FUNCTION_BLOCK ToteData
VAR_INPUT
	
END_VAR
VAR_OUTPUT
END_VAR
VAR_IN_OUT
	
END_VAR
VAR
	status	: ToteStatus:= ToteStatus.UNKNOWN;
	barcode	: STRING	:= '';
	barcode_validation	: BarcodeVerificationResult	:= BarcodeVerificationResult.UNVERIFIED;
	bag_status_0	: BagStatus;
	bag_status_1	: BagStatus;
	bag_opening_status_0	: BagOpeningStatus;
	bag_opening_status_1	: BagOpeningStatus;
	
	
END_VAR

PROPERTY _status : ToteStatus
GET
_status	:= status;
END_GET
SET

status	:= _status;
END_SET
END_PROPERTY

END_FUNCTION_BLOCK

(* stored: Version 1.1.0.1, ProductVersion 3.1.4024.12
   POU ToteData: Id {b550ec73-9a62-494f-ac6c-bd7075901bc6}, SpecialFunc None
   Property _status: Id {a57875de-fbad-45fa-9732-3f1850ab8f1a}
   Get Get: Id {19b59cf0-1b19-4941-80c4-ff7998d54d48}
   Set Set: Id {ed0320b0-d73b-42d0-8281-19a64b70d771} *)
